// Mitsubishi GX Works2 project: p3-1   PLC: FX3G

// global labels: Global1
VAR_GLOBAL
  Help_Lamp_1 AT M7 : BOOL;
  Stop_condition AT M8 : BOOL;
  Flickering_Light_1 AT M4 : BOOL;
  Timer_Value_1 AT TS0 : BOOL;
  Flickering_Timer_1 AT TC0 : BOOL;
END_VAR
VAR_GLOBAL CONSTANT
  Flickering_constant : INT := 5;
END_VAR
VAR_GLOBAL
  Flickering_Light_2 AT M5 : BOOL;
  Flickering_Timer_2 AT TC1 : BOOL;
  Timer_Value_2 AT TS1 : BOOL;
  Flickering_Light_OFF AT M6 : BOOL;
  StartCounter AT CC0 : BOOL;
END_VAR
VAR_GLOBAL CONSTANT
  CounterStart : INT := 1;
END_VAR
VAR_GLOBAL
  init_WorkDay AT X007 : BOOL;
  LoadMaterials AT CS0 : BOOL;
END_VAR
VAR_GLOBAL CONSTANT
  init_Cream : REAL := 700;
  init_Chocolate : REAL := 500;
  init_Biscuit : REAL := 100;
END_VAR
VAR_GLOBAL
  inventory_Cream AT D1100 : REAL;
END_VAR
VAR_GLOBAL CONSTANT
  minimum_Cream : REAL := 300;
END_VAR
VAR_GLOBAL
  inventory_Chocolate AT D1110 : REAL;
END_VAR
VAR_GLOBAL CONSTANT
  minimum_Chocolate : REAL := 240;
END_VAR
VAR_GLOBAL
  inventory_Biscuit AT D1120 : REAL;
END_VAR
VAR_GLOBAL CONSTANT
  minimum_Biscuit : REAL := 6;
END_VAR
VAR_GLOBAL
  valid_inventory AT M0 : BOOL;
  WorkDay_Lamp AT Y007 : BOOL;
  BreakHoldingSwich AT X007 : BOOL;
  Move_Cream_and_Biscuit AT X011 : BOOL;
  Fill_containers AT M1 : BOOL;
END_VAR
VAR_GLOBAL CONSTANT
  Fill_Cream : REAL := 300;
  Fill_Biscuit : REAL := 6;
  Zero : REAL;
END_VAR
VAR_GLOBAL
  Cream_Container AT D1130 : REAL;
  Biscuit_Container AT D1140 : REAL;
  Start_machine_A AT X010 : BOOL;
  Machine_A_ON AT M32 : BOOL;
  Eror_in_Machine_A AT X005 : BOOL;
  Sen_Crembo_in AT X001 : BOOL;
  Sen_Camera AT X004 : BOOL;
  Sen_30 AT X002 : BOOL;
  Sprinkling_Cream_ON AT Y004 : BOOL;
  Sen_15 AT X003 : BOOL;
  Stop_Flickering AT TS4 : BOOL;
  Timer_1 AT TC4 : BOOL;
END_VAR
VAR_GLOBAL CONSTANT
  Moving_Crembo_Time : INT := 40;
END_VAR
VAR_GLOBAL
  Lamp_0 AT Y000 : BOOL;
  Lamp_1 AT Y001 : BOOL;
  BUTTON AT X006 : BOOL;
  analog_value_set AT M8 : BOOL;
END_VAR
VAR_GLOBAL CONSTANT
  Condition1 : REAL := 5;
  one_layer : REAL := 120;
END_VAR
VAR_GLOBAL
  Chocolate_dipping_Container AT D1150 : REAL;
  dipping_timer AT TC3 : BOOL;
END_VAR
VAR_GLOBAL CONSTANT
  timer_5 : INT := 50;
END_VAR
VAR_GLOBAL
  Y7_Lamp AT Y007 : BOOL;
  Fs AT X010 : BOOL;
  read_analog AT X006 : BOOL;
  light AT Y011 : BOOL;
  dip_counter AT CC3 : BOOL;
END_VAR
VAR_GLOBAL CONSTANT
  Counterdip : INT := 1;
END_VAR
VAR_GLOBAL
  CON_1 AT M9 : BOOL;
END_VAR
VAR_GLOBAL CONSTANT
  Condition2 : REAL := 5;
  Two_layers : REAL := 240;
END_VAR
VAR_GLOBAL
  CON_2 AT M10 : BOOL;
  dipping_light AT Y003 : BOOL;
  dip_timer AT TS3 : BOOL;
  dipped AT M11 : BOOL;
  Start_Packing AT X000 : BOOL;
END_VAR
VAR_GLOBAL CONSTANT
  const_packing : INT := 5;
END_VAR
VAR_GLOBAL
  Packing_Counter AT CC1 : BOOL;
  Packing_Output AT CS1 : BOOL;
  Packing_Lamp AT Y002 : BOOL;
  Stop_Packing AT X000 : BOOL;
  Stop_Packing_Counter AT CC2 : BOOL;
END_VAR
VAR_GLOBAL CONSTANT
  const_packing_stop : INT := 6;
END_VAR
VAR_GLOBAL
  Stop_Packing_Lamp AT CS2 : BOOL;
END_VAR
VAR_GLOBAL CONSTANT
  const_Crembo : INT := 240;
END_VAR
VAR_GLOBAL
  analog_output AT D8282 : INT;
  iteration_Finished AT M2 : BOOL;
  End_day AT M3 : BOOL;
  Timer_2 AT TC5 : BOOL;
  Stop_Flickering_2 AT TS5 : BOOL;
END_VAR
VAR_GLOBAL CONSTANT
  Day_off_const : INT := 30;
END_VAR
VAR_GLOBAL
  Y7_Lamp_OFF AT M12 : BOOL;
  End_day_timer AT M13 : BOOL;
  lampFlickering_Light_21 AT M5 : BOOL;
  lampFlickering_Light_2 AT M5 : BOOL;
  blinking_Counter AT CC4 : BOOL;
END_VAR
VAR_GLOBAL CONSTANT
  const_blinking_Off : INT := 3;
END_VAR
VAR_GLOBAL
  inventory_initiation AT M14 : BOOL;
  Reset_Timers_ON AT M15 : BOOL;
  Reset_Counters_ON AT M16 : BOOL;
  Reset_Registors_ON AT M31 : BOOL;
  ready_to_start_new_iteration AT M17 : BOOL;
  Reset_Lamps_ON AT M18 : BOOL;
  analog_input_value AT D1170 : REAL;
  analog_input_1 AT D8280 : INT;
END_VAR
VAR_GLOBAL CONSTANT
  constAuto : REAL := 400;
END_VAR
VAR_GLOBAL
  Reset_day_ON AT M19 : BOOL;
  day_ON AT M20 : BOOL;
  True_1 AT M21 : BOOL;
  True_2 AT M22 : BOOL;
  True_3 AT M23 : BOOL;
  Help_Lamp_2 AT M24 : BOOL;
  out_of_stock AT M25 : BOOL;
  End_of_packaging AT M26 : BOOL;
  Stock_stop AT M27 : BOOL;
  dip_help AT M28 : BOOL;
  greater AT M29 : BOOL;
  isLower AT M30 : BOOL;
  rst_timer AT TC6 : BOOL;
  end_dip AT TS6 : BOOL;
  Enough_cream AT M33 : BOOL;
  Enough_biscuits AT M34 : BOOL;
  total_crembos AT D1160 : INT;
END_VAR
VAR_GLOBAL CONSTANT
  const_10 : REAL := 10;
END_VAR

// task Task_01 (event TRUE, interval 0, priority 31): POU_01

PROGRAM POU_01
VAR
  lower : BOOL;
END_VAR
(* structured ladder/FBD written out as ST: instructions are called as NAME(EN, inputs, outputs); _pN, _eN, _tN stand for wires *)
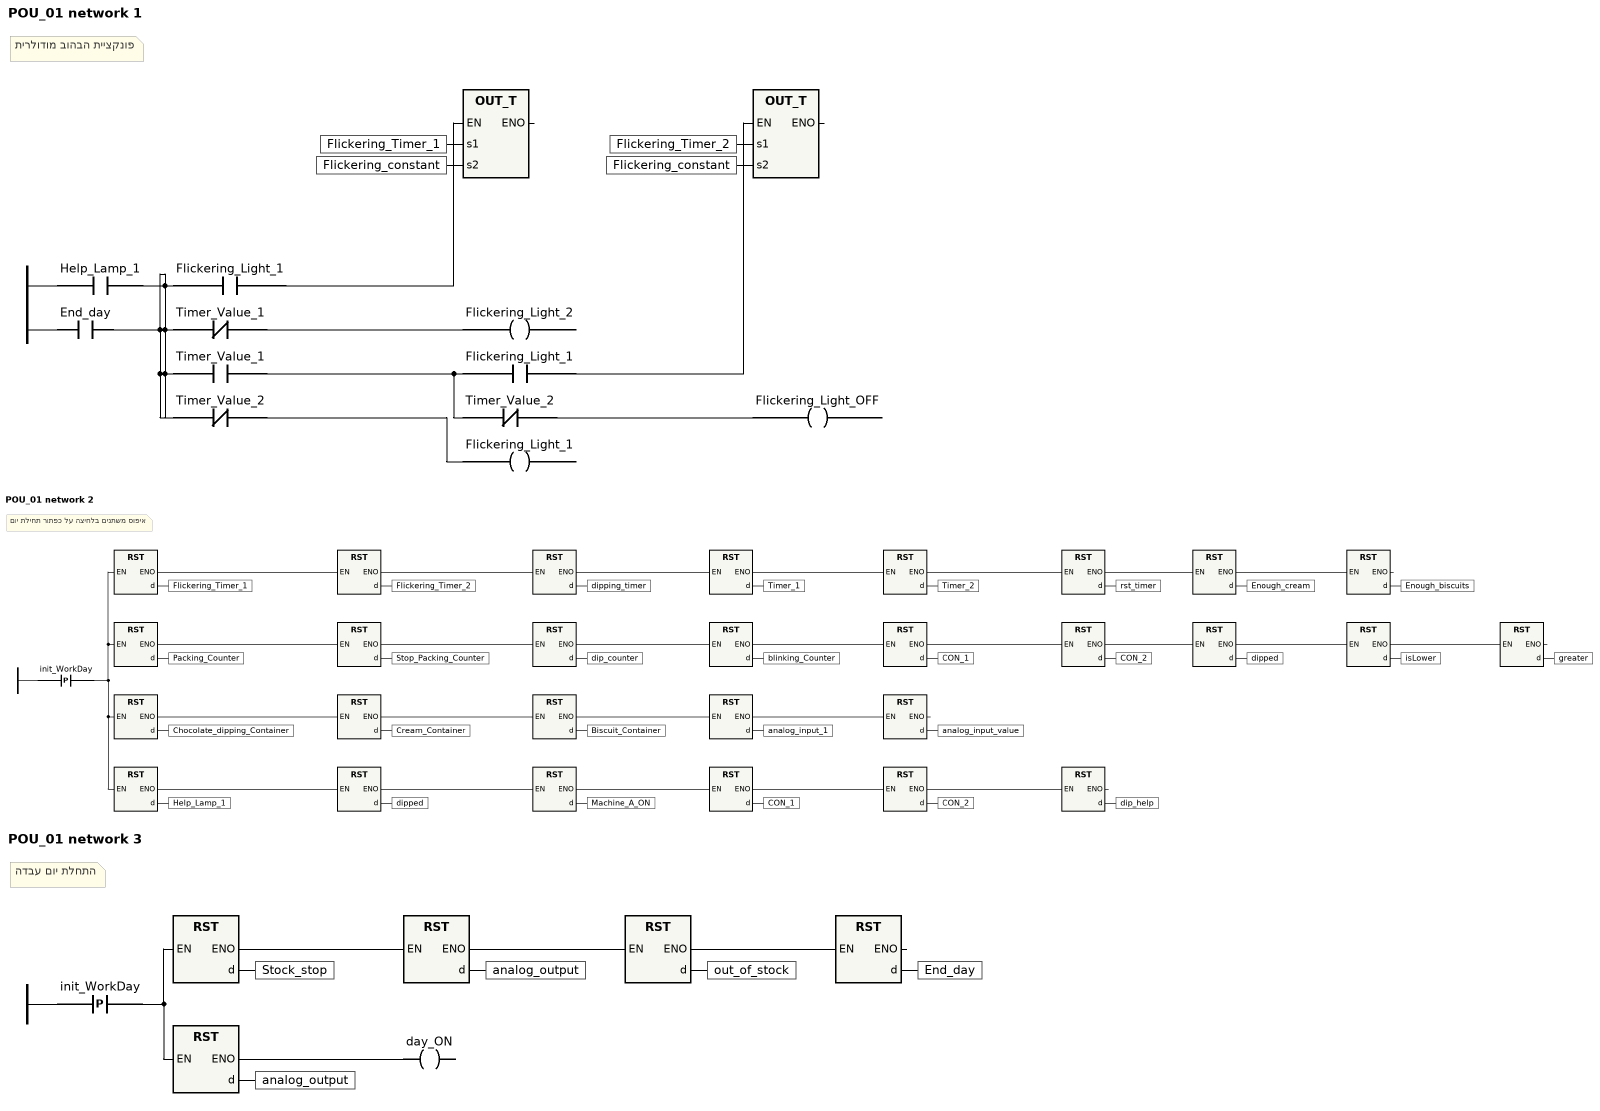
(* network 1 *)
(* פונקציית הבהוב מודולרית *)
_p1 := Help_Lamp_1 OR End_day;
OUT_T(_p1 AND Flickering_Light_1, Flickering_Timer_1, Flickering_constant);
Flickering_Light_2 := _p1 AND NOT Timer_Value_1;
_p2 := _p1 AND Timer_Value_1;
OUT_T(_p2 AND Flickering_Light_1, Flickering_Timer_2, Flickering_constant);
Flickering_Light_OFF := _p2 AND NOT Timer_Value_2;
Flickering_Light_1 := _p1 AND NOT Timer_Value_2;
(* network 2 *)
(* איפוס משתנים בלחיצה על כפתור תחילת יום *)
_p1 := LDP(TRUE, init_WorkDay);
_e2 := RST(_p1, Flickering_Timer_1);
_e3 := RST(_e2, Flickering_Timer_2);
_e4 := RST(_e3, dipping_timer);
_e5 := RST(_e4, Timer_1);
_e6 := RST(_e5, Timer_2);
_e7 := RST(_e6, rst_timer);
_e8 := RST(_e7, Enough_cream);
RST(_e8, Enough_biscuits);
_e9 := RST(_p1, Packing_Counter);
_e10 := RST(_e9, Stop_Packing_Counter);
_e11 := RST(_e10, dip_counter);
_e12 := RST(_e11, blinking_Counter);
_e13 := RST(_e12, CON_1);
_e14 := RST(_e13, CON_2);
_e15 := RST(_e14, dipped);
_e16 := RST(_e15, isLower);
RST(_e16, greater);
_e17 := RST(_p1, Chocolate_dipping_Container);
_e18 := RST(_e17, Cream_Container);
_e19 := RST(_e18, Biscuit_Container);
_e20 := RST(_e19, analog_input_1);
RST(_e20, analog_input_value);
_e21 := RST(_p1, Help_Lamp_1);
_e22 := RST(_e21, dipped);
_e23 := RST(_e22, Machine_A_ON);
_e24 := RST(_e23, CON_1);
_e25 := RST(_e24, CON_2);
RST(_e25, dip_help);
(* network 3 *)
(* התחלת יום עבדה *)
_p1 := LDP(TRUE, init_WorkDay);
_e2 := RST(_p1, Stock_stop);
_e3 := RST(_e2, analog_output);
_e4 := RST(_e3, out_of_stock);
RST(_e4, End_day);
_e5 := RST(_p1, analog_output);
day_ON := _e5;
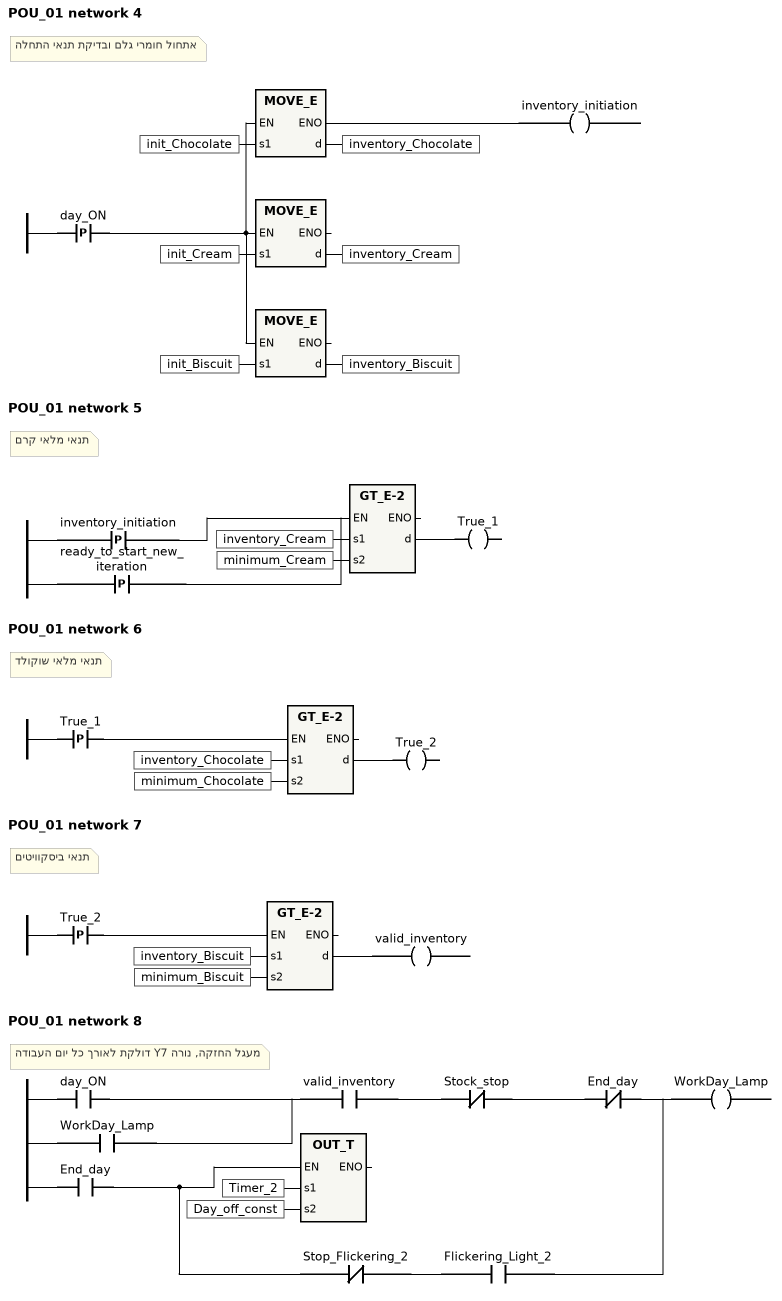
(* network 4 *)
(* אתחול חומרי גלם ובדיקת תנאי התחלה *)
_p1 := LDP(TRUE, day_ON);
MOVE_E(_p1, init_Cream, inventory_Cream);
_e2 := MOVE_E(_p1, init_Chocolate, inventory_Chocolate);
inventory_initiation := _e2;
MOVE_E(_p1, init_Biscuit, inventory_Biscuit);
(* network 5 *)
(* תנאי מלאי קרם *)
GT_E(LDP(TRUE, inventory_initiation) OR LDP(TRUE, ready_to_start_new_iteration), inventory_Cream, minimum_Cream, _t1);
True_1 := _t1;
(* network 6 *)
(* תנאי מלאי שוקולד *)
GT_E(LDP(TRUE, True_1), inventory_Chocolate, minimum_Chocolate, _t1);
True_2 := _t1;
(* network 7 *)
(* תנאי ביסקוויטים *)
GT_E(LDP(TRUE, True_2), inventory_Biscuit, minimum_Biscuit, _t1);
valid_inventory := _t1;
(* network 8 *)
(* מעגל החזקה, נורה Y7 דולקת לאורך כל יום העבודה *)
WorkDay_Lamp := ((((day_ON OR WorkDay_Lamp) AND valid_inventory) AND NOT Stock_stop) AND NOT End_day) OR (End_day AND NOT Stop_Flickering_2 AND Flickering_Light_2);
OUT_T(End_day, Timer_2, Day_off_const);
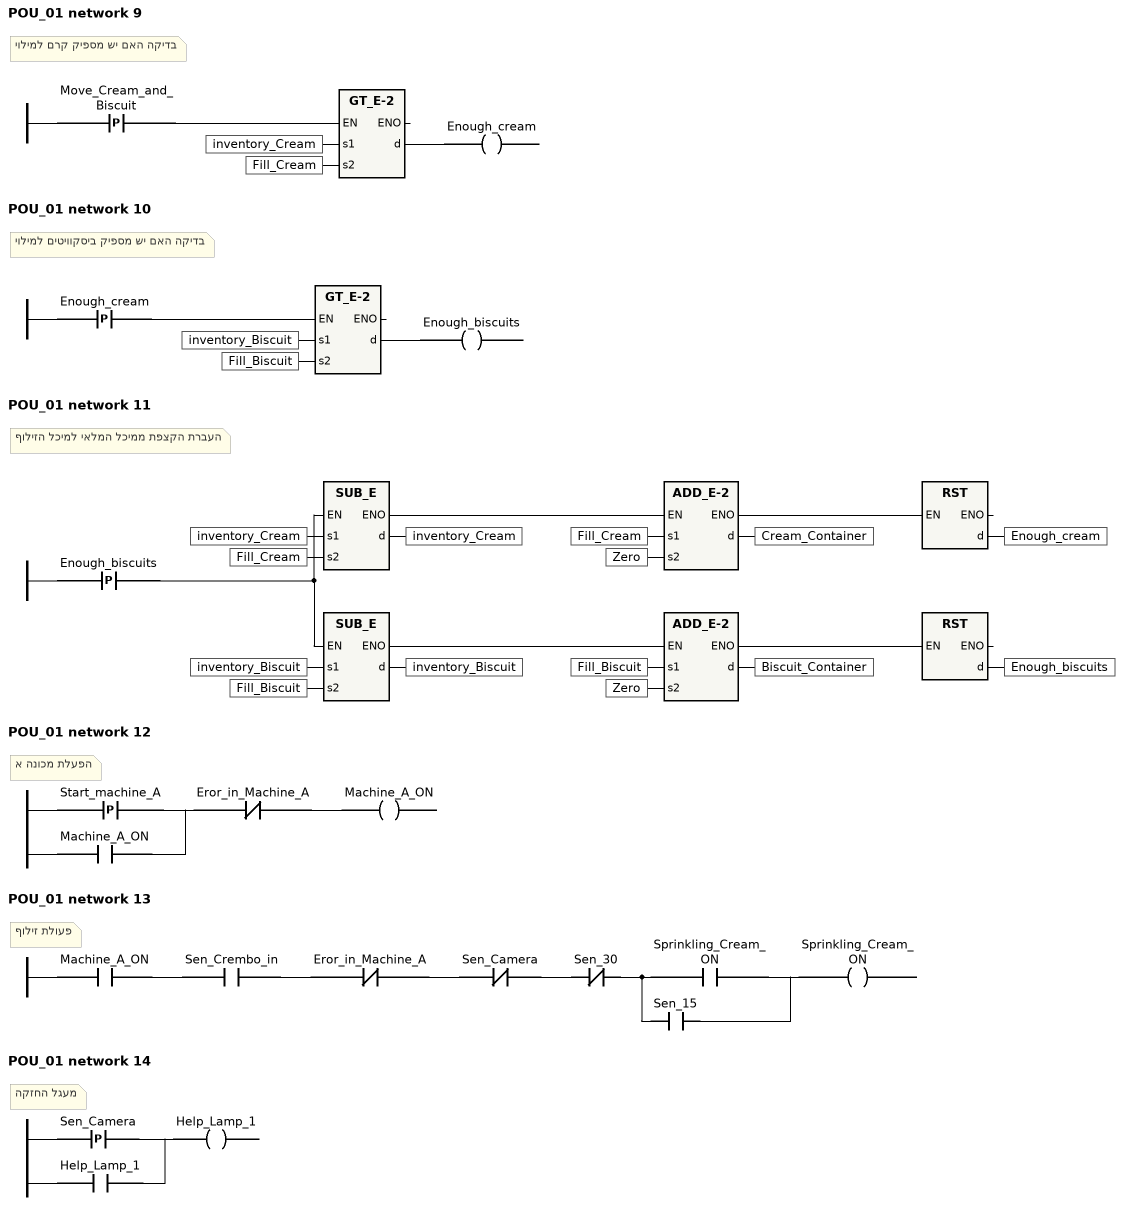
(* network 9 *)
(* בדיקה האם יש מספיק קרם למילוי *)
GT_E(LDP(TRUE, Move_Cream_and_Biscuit), inventory_Cream, Fill_Cream, _t1);
Enough_cream := _t1;
(* network 10 *)
(* בדיקה האם יש מספיק ביסקוויטים למילוי *)
GT_E(LDP(TRUE, Enough_cream), inventory_Biscuit, Fill_Biscuit, _t1);
Enough_biscuits := _t1;
(* network 11 *)
(* העברת הקצפת ממיכל המלאי למיכל הזילוף *)
_p1 := LDP(TRUE, Enough_biscuits);
_e2 := SUB_E(_p1, inventory_Cream, Fill_Cream, inventory_Cream);
_e3 := ADD_E(_e2, Fill_Cream, Zero, Cream_Container);
RST(_e3, Enough_cream);
_e4 := SUB_E(_p1, inventory_Biscuit, Fill_Biscuit, inventory_Biscuit);
_e5 := ADD_E(_e4, Fill_Biscuit, Zero, Biscuit_Container);
RST(_e5, Enough_biscuits);
(* network 12 *)
(* הפעלת מכונה א *)
Machine_A_ON := (LDP(TRUE, Start_machine_A) OR Machine_A_ON) AND NOT Eror_in_Machine_A;
(* network 13 *)
(* פעולת זילוף *)
_p1 := Machine_A_ON AND Sen_Crembo_in AND NOT Eror_in_Machine_A AND NOT Sen_Camera AND NOT Sen_30;
Sprinkling_Cream_ON := (_p1 AND Sprinkling_Cream_ON) OR (_p1 AND Sen_15);
(* network 14 *)
(* מעגל החזקה *)
Help_Lamp_1 := LDP(TRUE, Sen_Camera) OR Help_Lamp_1;
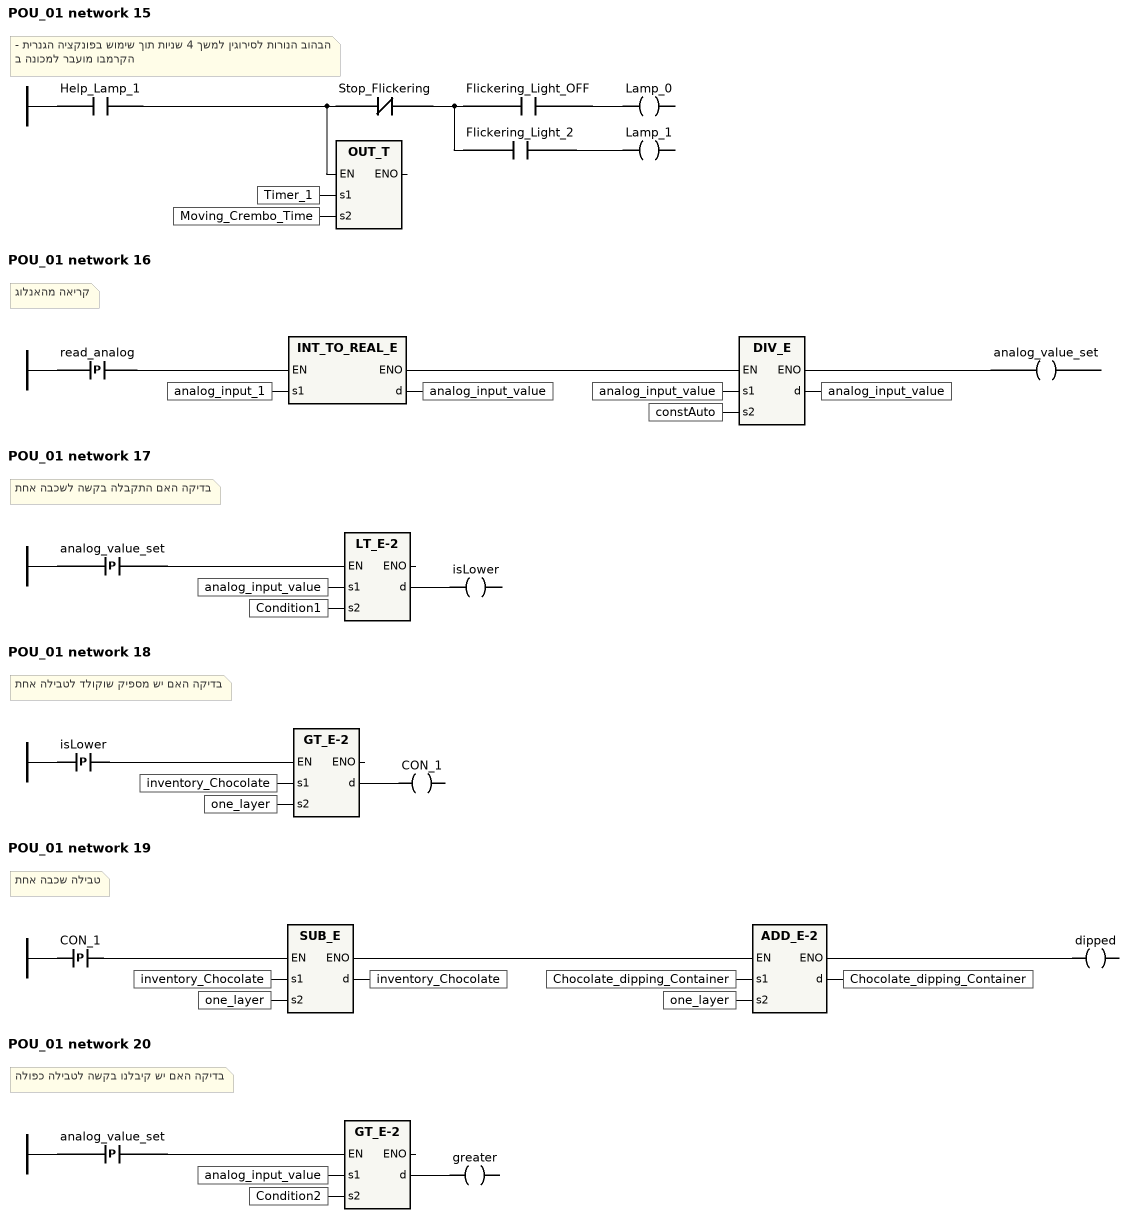
(* network 15 *)
(* הבהוב הנורות לסירוגין למשך 4 שניות תוך שימוש בפונקציה הגנרית - הקרמבו מועבר למכונה ב *)
_p1 := Help_Lamp_1 AND NOT Stop_Flickering;
Lamp_0 := _p1 AND Flickering_Light_OFF;
Lamp_1 := _p1 AND Flickering_Light_2;
OUT_T(Help_Lamp_1, Timer_1, Moving_Crembo_Time);
(* network 16 *)
(* קריאה מהאנלוג *)
_e1 := INT_TO_REAL_E(LDP(TRUE, read_analog), analog_input_1, analog_input_value);
_e2 := DIV_E(_e1, analog_input_value, constAuto, analog_input_value);
analog_value_set := _e2;
(* network 17 *)
(* בדיקה האם התקבלה בקשה לשכבה אחת *)
LT_E(LDP(TRUE, analog_value_set), analog_input_value, Condition1, _t1);
isLower := _t1;
(* network 18 *)
(* בדיקה האם יש מספיק שוקולד לטבילה אחת *)
GT_E(LDP(TRUE, isLower), inventory_Chocolate, one_layer, _t1);
CON_1 := _t1;
(* network 19 *)
(* טבילה שכבה אחת *)
_e1 := SUB_E(LDP(TRUE, CON_1), inventory_Chocolate, one_layer, inventory_Chocolate);
_e2 := ADD_E(_e1, Chocolate_dipping_Container, one_layer, Chocolate_dipping_Container);
dipped := _e2;
(* network 20 *)
(* בדיקה האם יש קיבלנו בקשה לטבילה כפולה *)
GT_E(LDP(TRUE, analog_value_set), analog_input_value, Condition2, _t1);
greater := _t1;
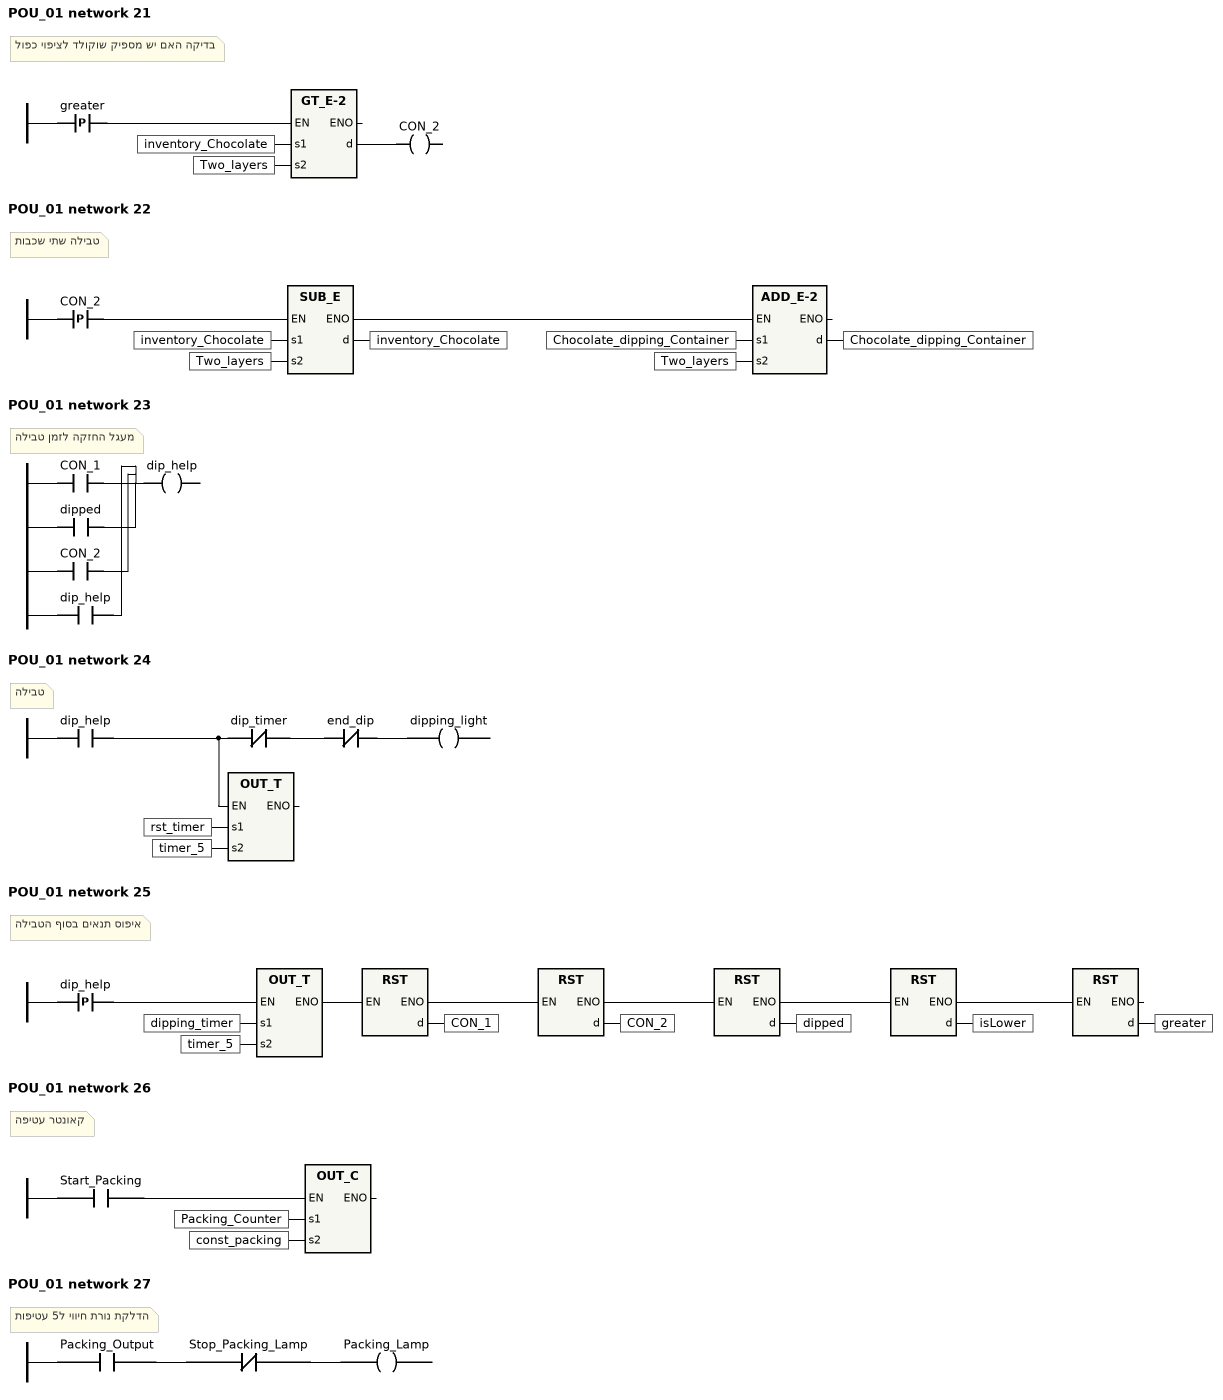
(* network 21 *)
(* בדיקה האם יש מספיק שוקולד לציפוי כפול *)
GT_E(LDP(TRUE, greater), inventory_Chocolate, Two_layers, _t1);
CON_2 := _t1;
(* network 22 *)
(* טבילה שתי שכבות *)
_e1 := SUB_E(LDP(TRUE, CON_2), inventory_Chocolate, Two_layers, inventory_Chocolate);
ADD_E(_e1, Chocolate_dipping_Container, Two_layers, Chocolate_dipping_Container);
(* network 23 *)
(* מעגל החזקה לזמן טבילה *)
dip_help := CON_1 OR dipped OR CON_2 OR dip_help;
(* network 24 *)
(* טבילה *)
dipping_light := dip_help AND NOT dip_timer AND NOT end_dip;
OUT_T(dip_help, rst_timer, timer_5);
(* network 25 *)
(* איפוס תנאים בסוף הטבילה *)
_e1 := OUT_T(LDP(TRUE, dip_help), dipping_timer, timer_5);
_e2 := RST(_e1, CON_1);
_e3 := RST(_e2, CON_2);
_e4 := RST(_e3, dipped);
_e5 := RST(_e4, isLower);
RST(_e5, greater);
(* network 26 *)
(* קאונטר עטיפה *)
OUT_C(Start_Packing, Packing_Counter, const_packing);
(* network 27 *)
(* הדלקת נורת חיווי ל5 עטיפות *)
Packing_Lamp := Packing_Output AND NOT Stop_Packing_Lamp;
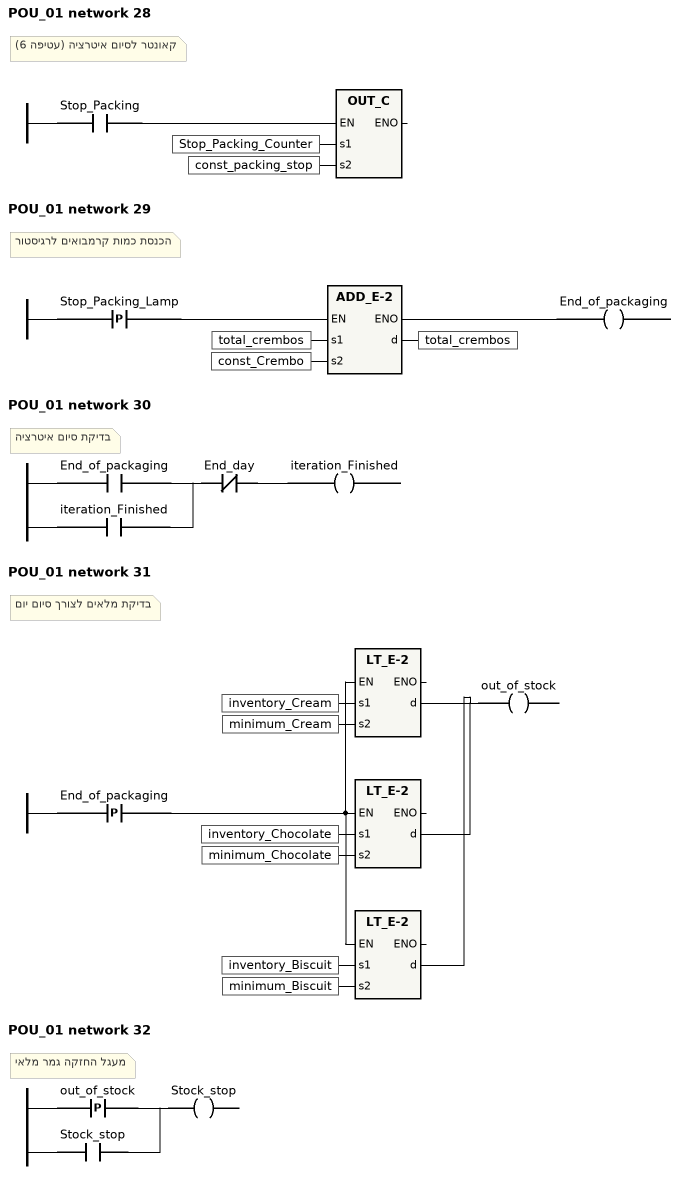
(* network 28 *)
(* קאונטר לסיום איטרציה (עטיפה 6) *)
OUT_C(Stop_Packing, Stop_Packing_Counter, const_packing_stop);
(* network 29 *)
(* הכנסת כמות קרמבואים לרגיסטור *)
_e1 := ADD_E(LDP(TRUE, Stop_Packing_Lamp), total_crembos, const_Crembo, total_crembos);
End_of_packaging := _e1;
(* network 30 *)
(* בדיקת סיום איטרציה *)
iteration_Finished := (End_of_packaging OR iteration_Finished) AND NOT End_day;
(* network 31 *)
(* בדיקת מלאים לצורך סיום יום *)
_p1 := LDP(TRUE, End_of_packaging);
LT_E(_p1, inventory_Cream, minimum_Cream, _t2);
LT_E(_p1, inventory_Chocolate, minimum_Chocolate, _t3);
LT_E(_p1, inventory_Biscuit, minimum_Biscuit, _t4);
out_of_stock := _t2 OR _t3 OR _t4;
(* network 32 *)
(* מעגל החזקה גמר מלאי *)
Stock_stop := LDP(TRUE, out_of_stock) OR Stock_stop;
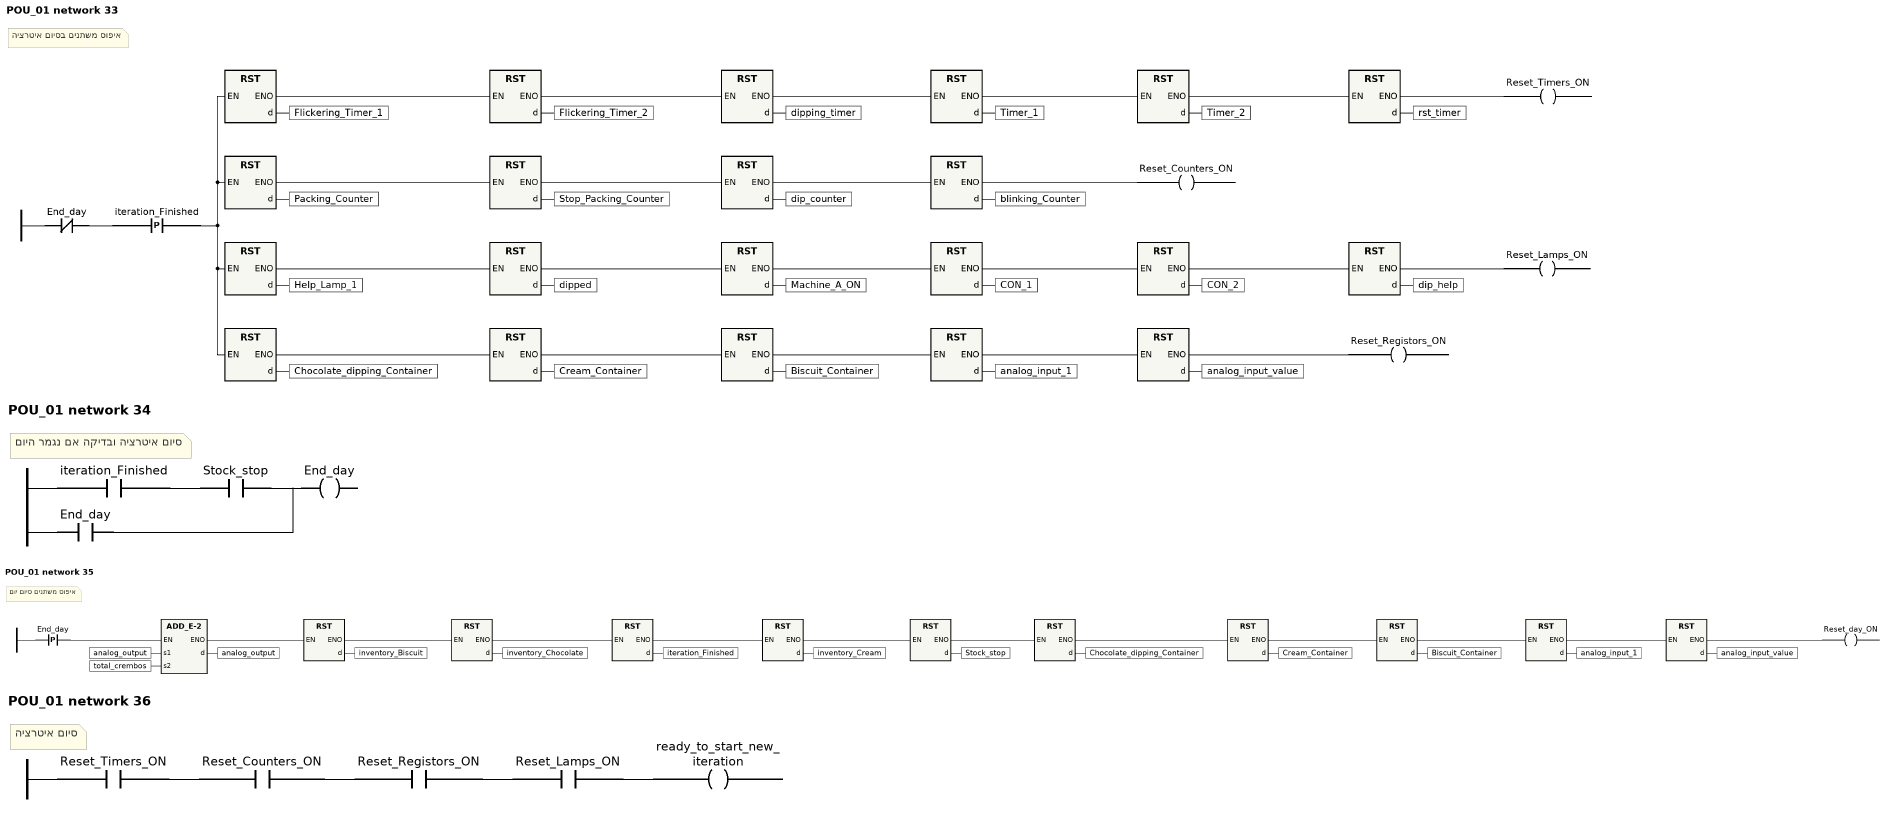
(* network 33 *)
(* איפוס משתנים בסיום איטרציה *)
_p1 := NOT End_day AND LDP(TRUE, iteration_Finished);
_e2 := RST(_p1, Flickering_Timer_1);
_e3 := RST(_e2, Flickering_Timer_2);
_e4 := RST(_e3, dipping_timer);
_e5 := RST(_e4, Timer_1);
_e6 := RST(_e5, Timer_2);
_e7 := RST(_e6, rst_timer);
Reset_Timers_ON := _e7;
_e8 := RST(_p1, Packing_Counter);
_e9 := RST(_e8, Stop_Packing_Counter);
_e10 := RST(_e9, dip_counter);
_e11 := RST(_e10, blinking_Counter);
Reset_Counters_ON := _e11;
_e12 := RST(_p1, Chocolate_dipping_Container);
_e13 := RST(_e12, Cream_Container);
_e14 := RST(_e13, Biscuit_Container);
_e15 := RST(_e14, analog_input_1);
_e16 := RST(_e15, analog_input_value);
Reset_Registors_ON := _e16;
_e17 := RST(_p1, Help_Lamp_1);
_e18 := RST(_e17, dipped);
_e19 := RST(_e18, Machine_A_ON);
_e20 := RST(_e19, CON_1);
_e21 := RST(_e20, CON_2);
_e22 := RST(_e21, dip_help);
Reset_Lamps_ON := _e22;
(* network 34 *)
(* סיום איטרציה ובדיקה אם נגמר היום *)
End_day := (iteration_Finished AND Stock_stop) OR End_day;
(* network 35 *)
(* איפוס משתנים סיום יום *)
_e1 := ADD_E(LDP(TRUE, End_day), analog_output, total_crembos, analog_output);
_e2 := RST(_e1, inventory_Biscuit);
_e3 := RST(_e2, inventory_Chocolate);
_e4 := RST(_e3, iteration_Finished);
_e5 := RST(_e4, inventory_Cream);
_e6 := RST(_e5, Stock_stop);
_e7 := RST(_e6, Chocolate_dipping_Container);
_e8 := RST(_e7, Cream_Container);
_e9 := RST(_e8, Biscuit_Container);
_e10 := RST(_e9, analog_input_1);
_e11 := RST(_e10, analog_input_value);
Reset_day_ON := _e11;
(* network 36 *)
(* סיום איטרציה *)
ready_to_start_new_iteration := Reset_Timers_ON AND Reset_Counters_ON AND Reset_Registors_ON AND Reset_Lamps_ON;
END_PROGRAM
